{attribute 'GeneratedUsingTerminal: EK1100-0000-0018'}
{attribute addProperty BoxType "EK1100-0000-0018"}
{attribute addProperty Id "Term_2_EL1809EL1809_32157CFD20"}
{attribute addProperty CRC "3324839725"}
{attribute addProperty Size "20"}
TYPE Term_1_EK1100_C62D072D EXTENDS EK1100_1FC0878B :
STRUCT
	{attribute addProperty Name "Term 2 (EL1809)"}
	{attribute addProperty PreviousPort "Term 1 (EK1100) : B"}
	Term_2_EL1809 : EL1809_32157CFD;
END_STRUCT
END_TYPE

(* stored: Version 1.2.0.0, ProductVersion 3.1.4024.11
   DUT Term_1_EK1100_C62D072D: Id {417ae2ea-4980-4c30-9b7c-25a6e67f94f3} *)
